Yaskawa INFORM job: ROS_R1.JBI

/JOB
//NAME ROS_R1
//POS
///NPOS 0,0,0,0,0,0
//INST
///DATE 2014/06/16 09:25
///ATTR SC,RW
///GROUP1 RB1
NOP
DOUT OT#(890) OFF
DOUT OT#(889) OFF
TIMER T=0.05
SKILLSND "ROS-START"
TSYNC 1
DOUT OT#(889) ON
WAIT OT#(890)=ON
DOUT OT#(889) OFF
DOUT OT#(890) OFF
SKILLSND "ROS-STOP"
END
